(********************* G.D S.p.A. - Technical Department ***********************************
Date        Version Author      	Description             
----------  ------- ----------- 	--------------------------------------------------------
2019/04/23	0000.01	G.Cera			Creation of the POU

DESCRIPTION:
Manager of the application status high. it is called by highest speed task


NOTES:

********************************************************************************************)
PROGRAM application_status_manager_highest
VAR

END_VAR

VAR_OUTPUT

END_VAR

IF g_application_status=APPLICATION_STATUS_1ST_POWERUP_ABSOLUTE
THEN
   	g_application_status_1st_powerup_high_absolute:=TRUE;
END_IF

IF g_application_status=APPLICATION_STATUS_1ST_POWERUP
THEN
   	g_application_status_1st_powerup_high:=TRUE;
END_IF

IF g_application_status=APPLICATION_STATUS_2ND_POWERUP
THEN
   	g_application_status_2nd_powerup_high:=TRUE;
END_IF

IF g_application_status=APPLICATION_STATUS_3RD_POWERUP
THEN
   	g_application_status_3rd_powerup_high:=TRUE;
END_IF;

END_PROGRAM

(* stored: Version 1.1.0.1, ProductVersion 3.1.4022.12
   POU application_status_manager_highest: Id {a19a63b5-d343-4870-ac26-75b26e3f9b9b}, SpecialFunc None *)
